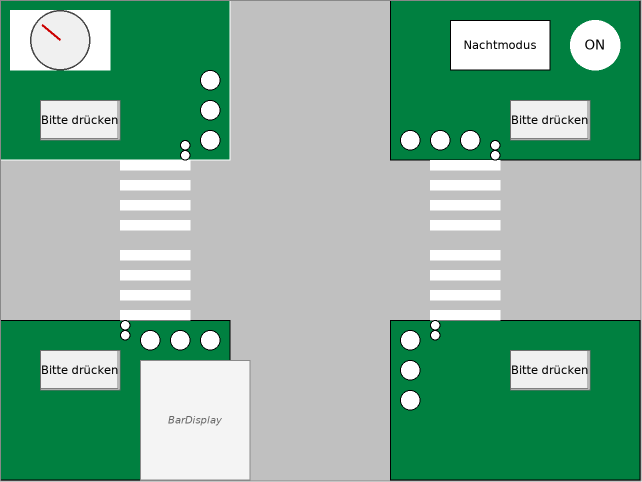
VISUALIZATION Kreuzung  // 642x482
    Rectangle (230,0 160x480)
    Rectangle (0,160 640x160)
    Rectangle (0,0 230x160)
    Rectangle (390,0 250x160)
        tap MAIN.bON
    Rectangle (390,320 250x160)
    Rectangle (0,320 230x160)
    Polyline (230,0)
    Polyline (630,160)
    Polyline (230,480)
    Polyline (630,320)
    Ellipse (200,330 20x20), colour toggle: MAIN.bWO_rot
    Ellipse (170,330 20x20), colour toggle: MAIN.bWO_orange
    Ellipse (140,330 20x20), colour toggle: MAIN.bWO_gruen
    Ellipse (400,360 20x20), colour toggle: MAIN.bNS_orange
    Ellipse (400,330 20x20), colour toggle: MAIN.bNS_rot
    Ellipse (460,130 20x20), colour toggle: MAIN.bWO_gruen
    Ellipse (430,130 20x20), colour toggle: MAIN.bWO_orange
    Ellipse (400,130 20x20), colour toggle: MAIN.bWO_rot
    Ellipse (400,390 20x20), colour toggle: MAIN.bNS_gruen
    Ellipse (200,130 20x20), colour toggle: MAIN.bNS_rot
    Ellipse (200,100 20x20), colour toggle: MAIN.bNS_orange
    Ellipse (200,70 20x20), colour toggle: MAIN.bNS_gruen
    Polyline (20,240)
    Polyline (60,240)
    Polyline (100,240)
    Polyline (140,240)
    Polyline (180,240)
    Polyline (220,240)
    Polyline (460,240)
    Polyline (540,240)
    Polyline (500,240)
    Polyline (580,240)
    Polyline (620,240)
    Polyline (310,340)
    Polyline (310,380)
    Polyline (310,420)
    Polyline (310,460)
    Polyline (310,480)
    Polyline (310,160)
    Polyline (310,120)
    Polyline (310,80)
    Polyline (310,40)
    Polyline (310,10)
    Ellipse (570,20 50x50), "ON", colour toggle: MAIN.bON
        toggle MAIN.bON
    Rectangle (10,10 100x60)
    Meter (10,10 100x60), value: MAIN.iPhase, scale format: %.1f, scale 0..4
    Rectangle (430,200 70x10)
    Rectangle (430,250 70x10)
    Rectangle (430,180 70x10)
    Rectangle (430,310 70x10)
    Rectangle (430,220 70x10)
    Rectangle (430,270 70x10)
    Rectangle (430,290 70x10)
    Rectangle (430,160 70x10)
    Polyline (420,240)
    Rectangle (120,200 70x10)
    Rectangle (120,250 70x10)
    Rectangle (120,180 70x10)
    Rectangle (120,310 70x10)
    Rectangle (120,220 70x10)
    Rectangle (120,270 70x10)
    Rectangle (120,290 70x10)
    Rectangle (120,160 70x10)
    Ellipse (120,330 10x10), colour toggle: MAIN.bFGNS_rot
    Ellipse (120,320 10x10), colour toggle: MAIN.bFGNS_gruen
    Ellipse (180,150 10x10), colour toggle: MAIN.bFGNS_gruen
    Ellipse (180,140 10x10), colour toggle: MAIN.bFGNS_rot
    Ellipse (430,330 10x10), colour toggle: MAIN.bFGNS_rot
    Ellipse (430,320 10x10), colour toggle: MAIN.bFGNS_gruen
    Ellipse (490,150 10x10), colour toggle: MAIN.bFGNS_gruen
    Ellipse (490,140 10x10), colour toggle: MAIN.bFGNS_rot
    Button (510,350 80x40), "Bitte drücken", pressed state: MAIN.bFG
        toggle MAIN.bFG
    Button (40,100 80x40), "Bitte drücken", pressed state: MAIN.bFG
        toggle MAIN.bFG
    Button (510,100 80x40), "Bitte drücken", pressed state: MAIN.bFG
        toggle MAIN.bFG
    Button (40,350 80x40), "Bitte drücken", pressed state: MAIN.bFG
        toggle MAIN.bFG
    RoundedRectangle (450,20 100x50), "Nachtmodus", colour toggle: MAIN.bNacht
        toggle MAIN.bNacht
    Rectangle (150,360 70x120)
    BarDisplay (140,360 110x120), value: MAIN.iPhase, scale format: %.1f, scale 0..4
END_VISUALIZATION

(* stored: Version 1.1.0.1, ProductVersion 3.1.4024.0
   Visu Kreuzung: Id {663b522c-a0dc-4b21-9db8-16638f0d0a2c} *)
